FUNCTION_BLOCK FB_Regelschuif
VAR_INPUT
END_VAR
VAR_OUTPUT
END_VAR
VAR
END_VAR

END_FUNCTION_BLOCK

(* stored: Version 1.1.0.1, ProductVersion 3.1.4026.8
   POU FB_Regelschuif: Id {197a057b-7e77-4001-97d3-497a9b935830}, SpecialFunc None *)
